ABB RobotStudio station: Solution15.rsstn

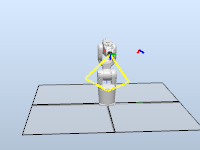
Station Solution15 (saved by RobotStudio 21.4.9700.0)
Controller IRB1200_7_70_1_LONG
  mechanical unit ROB_1: IRB1200_7_70_STD_03, 6 joints, base frame (0, 0, 0) mm
Layout (positions relative to the parent item):
  - IRB1200_7_70_STD_03 [mechanism, from Robots\IRB1200_7_70_STD_03.rslib] at (0, 0, 0) mm; joint values [-0.0012, -0.0017, 0.0867, -0.015, -0.085, 0.0148] (rad or m)
Targets, tools, work objects and paths stored in the station, written as RAPID:
! task T_ROB1
MODULE Module1
  CONST robtarget Target_10:=[[422.014082513,0,750.099998965],[0.499999994,0,0.866025407,0],[0,0,0,0],[9E+09,9E+09,9E+09,9E+09,9E+09,9E+09]];
  CONST robtarget Target_20:=[[116.600967602,405.58611933,750.099998965],[0.399420887,-0.520949955,0.691817281,0.300770592],[0,0,-1,0],[9E+09,9E+09,9E+09,9E+09,9E+09,9E+09]];
  CONST jointtarget JointTarget_0:=[[-0.62,0.28,5.37,-6.22,-5.68,6.19],[9E+09,9E+09,9E+09,9E+09,9E+09,9E+09]];
  CONST jointtarget JointTarget_1:=[[-1.23,0.35,5.9,-11.16,-6.37,11.09],[9E+09,9E+09,9E+09,9E+09,9E+09,9E+09]];
  CONST jointtarget JointTarget_2:=[[-1.84,0.44,6.41,-15.11,-7.09,15],[9E+09,9E+09,9E+09,9E+09,9E+09,9E+09]];
  CONST jointtarget JointTarget_3:=[[-2.46,0.53,6.92,-18.33,-7.84,18.17],[9E+09,9E+09,9E+09,9E+09,9E+09,9E+09]];
  CONST jointtarget JointTarget_4:=[[-3.07,0.64,7.41,-20.97,-8.61,20.76],[9E+09,9E+09,9E+09,9E+09,9E+09,9E+09]];
  CONST jointtarget JointTarget_5:=[[-3.69,0.77,7.89,-23.18,-9.4,22.9],[9E+09,9E+09,9E+09,9E+09,9E+09,9E+09]];
  CONST jointtarget JointTarget_6:=[[-4.3,0.9,8.35,-25.05,-10.2,24.7],[9E+09,9E+09,9E+09,9E+09,9E+09,9E+09]];
  CONST jointtarget JointTarget_7:=[[-4.91,1.05,8.8,-26.64,-11,26.22],[9E+09,9E+09,9E+09,9E+09,9E+09,9E+09]];
  CONST jointtarget JointTarget_8:=[[-5.52,1.21,9.25,-28.02,-11.81,27.52],[9E+09,9E+09,9E+09,9E+09,9E+09,9E+09]];
  CONST jointtarget JointTarget_9:=[[-6.13,1.39,9.67,-29.23,-12.63,28.63],[9E+09,9E+09,9E+09,9E+09,9E+09,9E+09]];
  CONST jointtarget JointTarget_11:=[[-7.34,1.78,10.5,-31.22,-14.27,30.43],[9E+09,9E+09,9E+09,9E+09,9E+09,9E+09]];
  CONST jointtarget JointTarget_12:=[[-7.95,1.99,10.89,-32.06,-15.09,31.16],[9E+09,9E+09,9E+09,9E+09,9E+09,9E+09]];
  CONST jointtarget JointTarget_13:=[[-8.55,2.21,11.27,-32.81,-15.92,31.8],[9E+09,9E+09,9E+09,9E+09,9E+09,9E+09]];
  CONST jointtarget JointTarget_14:=[[-9.15,2.45,11.63,-33.5,-16.74,32.36],[9E+09,9E+09,9E+09,9E+09,9E+09,9E+09]];
  CONST jointtarget JointTarget_15:=[[-9.75,2.7,11.99,-34.12,-17.57,32.86],[9E+09,9E+09,9E+09,9E+09,9E+09,9E+09]];
  CONST jointtarget JointTarget_16:=[[-10.34,2.97,12.33,-34.68,-18.39,33.29],[9E+09,9E+09,9E+09,9E+09,9E+09,9E+09]];
  CONST jointtarget JointTarget_17:=[[-10.94,3.24,12.66,-35.2,-19.22,33.67],[9E+09,9E+09,9E+09,9E+09,9E+09,9E+09]];
  CONST jointtarget JointTarget_18:=[[-11.53,3.53,12.97,-35.69,-20.04,34.01],[9E+09,9E+09,9E+09,9E+09,9E+09,9E+09]];
  CONST jointtarget JointTarget_19:=[[-12.12,3.83,13.27,-36.13,-20.86,34.3],[9E+09,9E+09,9E+09,9E+09,9E+09,9E+09]];
  CONST jointtarget JointTarget_21:=[[-13.29,4.47,13.84,-36.94,-22.49,34.79],[9E+09,9E+09,9E+09,9E+09,9E+09,9E+09]];
  CONST jointtarget JointTarget_22:=[[-13.87,4.8,14.11,-37.31,-23.3,34.99],[9E+09,9E+09,9E+09,9E+09,9E+09,9E+09]];
  CONST jointtarget JointTarget_23:=[[-14.45,5.15,14.36,-37.65,-24.11,35.16],[9E+09,9E+09,9E+09,9E+09,9E+09,9E+09]];
  CONST jointtarget JointTarget_24:=[[-15.02,5.51,14.6,-37.98,-24.91,35.3],[9E+09,9E+09,9E+09,9E+09,9E+09,9E+09]];
  CONST jointtarget JointTarget_25:=[[-15.6,5.88,14.82,-38.29,-25.72,35.43],[9E+09,9E+09,9E+09,9E+09,9E+09,9E+09]];
  CONST jointtarget JointTarget_26:=[[-16.17,6.27,15.04,-38.59,-26.51,35.53],[9E+09,9E+09,9E+09,9E+09,9E+09,9E+09]];
  CONST jointtarget JointTarget_27:=[[-16.73,6.66,15.23,-38.87,-27.3,35.61],[9E+09,9E+09,9E+09,9E+09,9E+09,9E+09]];
  CONST jointtarget JointTarget_28:=[[-17.29,7.07,15.42,-39.15,-28.09,35.68],[9E+09,9E+09,9E+09,9E+09,9E+09,9E+09]];
  CONST jointtarget JointTarget_29:=[[-17.85,7.48,15.6,-39.41,-28.88,35.74],[9E+09,9E+09,9E+09,9E+09,9E+09,9E+09]];
  CONST jointtarget JointTarget_30:=[[-18.41,7.91,15.76,-39.67,-29.65,35.78],[9E+09,9E+09,9E+09,9E+09,9E+09,9E+09]];
  CONST jointtarget JointTarget_31:=[[-18.96,8.35,15.9,-39.91,-30.43,35.8],[9E+09,9E+09,9E+09,9E+09,9E+09,9E+09]];
  CONST jointtarget JointTarget_32:=[[-19.51,8.8,16.04,-40.15,-31.19,35.82],[9E+09,9E+09,9E+09,9E+09,9E+09,9E+09]];
  CONST jointtarget JointTarget_33:=[[-20.05,9.26,16.16,-40.39,-31.95,35.82],[9E+09,9E+09,9E+09,9E+09,9E+09,9E+09]];
  CONST jointtarget JointTarget_34:=[[-20.6,9.72,16.27,-40.61,-32.71,35.81],[9E+09,9E+09,9E+09,9E+09,9E+09,9E+09]];
  CONST jointtarget JointTarget_35:=[[-21.13,10.2,16.36,-40.84,-33.46,35.8],[9E+09,9E+09,9E+09,9E+09,9E+09,9E+09]];
  CONST jointtarget JointTarget_36:=[[-21.67,10.69,16.44,-41.06,-34.2,35.77],[9E+09,9E+09,9E+09,9E+09,9E+09,9E+09]];
  CONST jointtarget JointTarget_37:=[[-22.19,11.19,16.51,-41.28,-34.93,35.74],[9E+09,9E+09,9E+09,9E+09,9E+09,9E+09]];
  CONST jointtarget JointTarget_38:=[[-22.72,11.7,16.56,-41.49,-35.66,35.7],[9E+09,9E+09,9E+09,9E+09,9E+09,9E+09]];
  CONST jointtarget JointTarget_39:=[[-23.24,12.21,16.6,-41.7,-36.38,35.65],[9E+09,9E+09,9E+09,9E+09,9E+09,9E+09]];
  CONST jointtarget JointTarget_40:=[[-23.76,12.74,16.63,-41.91,-37.1,35.6],[9E+09,9E+09,9E+09,9E+09,9E+09,9E+09]];
  CONST jointtarget JointTarget_41:=[[-24.27,13.27,16.65,-42.12,-37.8,35.54],[9E+09,9E+09,9E+09,9E+09,9E+09,9E+09]];
  CONST jointtarget JointTarget_42:=[[-24.78,13.81,16.65,-42.32,-38.5,35.48],[9E+09,9E+09,9E+09,9E+09,9E+09,9E+09]];
  CONST jointtarget JointTarget_43:=[[-25.29,14.36,16.64,-42.53,-39.19,35.41],[9E+09,9E+09,9E+09,9E+09,9E+09,9E+09]];
  CONST jointtarget JointTarget_44:=[[-25.79,14.92,16.61,-42.73,-39.87,35.34],[9E+09,9E+09,9E+09,9E+09,9E+09,9E+09]];
  CONST jointtarget JointTarget_45:=[[-26.28,15.49,16.57,-42.94,-40.55,35.26],[9E+09,9E+09,9E+09,9E+09,9E+09,9E+09]];
  CONST jointtarget JointTarget_46:=[[-26.78,16.06,16.52,-43.14,-41.21,35.18],[9E+09,9E+09,9E+09,9E+09,9E+09,9E+09]];
  CONST jointtarget JointTarget_47:=[[-27.26,16.64,16.45,-43.35,-41.87,35.1],[9E+09,9E+09,9E+09,9E+09,9E+09,9E+09]];
  CONST jointtarget JointTarget_48:=[[-27.75,17.23,16.37,-43.55,-42.51,35.02],[9E+09,9E+09,9E+09,9E+09,9E+09,9E+09]];
  CONST jointtarget JointTarget_49:=[[-28.23,17.82,16.28,-43.75,-43.15,34.93],[9E+09,9E+09,9E+09,9E+09,9E+09,9E+09]];
  CONST jointtarget JointTarget_50:=[[-28.7,18.42,16.18,-43.96,-43.78,34.84],[9E+09,9E+09,9E+09,9E+09,9E+09,9E+09]];
  CONST jointtarget JointTarget_51:=[[-29.17,19.03,16.06,-44.16,-44.4,34.76],[9E+09,9E+09,9E+09,9E+09,9E+09,9E+09]];
  CONST jointtarget JointTarget_52:=[[-29.64,19.65,15.93,-44.37,-45.01,34.66],[9E+09,9E+09,9E+09,9E+09,9E+09,9E+09]];
  CONST jointtarget JointTarget_53:=[[-30.1,20.27,15.78,-44.57,-45.61,34.57],[9E+09,9E+09,9E+09,9E+09,9E+09,9E+09]];
  CONST jointtarget JointTarget_54:=[[-30.56,20.89,15.62,-44.78,-46.21,34.48],[9E+09,9E+09,9E+09,9E+09,9E+09,9E+09]];
  CONST jointtarget JointTarget_55:=[[-31.02,21.52,15.45,-44.99,-46.79,34.39],[9E+09,9E+09,9E+09,9E+09,9E+09,9E+09]];
  CONST jointtarget JointTarget_56:=[[-31.47,22.16,15.27,-45.2,-47.36,34.3],[9E+09,9E+09,9E+09,9E+09,9E+09,9E+09]];
  CONST jointtarget JointTarget_57:=[[-31.91,22.8,15.07,-45.41,-47.92,34.21],[9E+09,9E+09,9E+09,9E+09,9E+09,9E+09]];
  CONST jointtarget JointTarget_58:=[[-32.35,23.44,14.86,-45.62,-48.48,34.12],[9E+09,9E+09,9E+09,9E+09,9E+09,9E+09]];
  CONST jointtarget JointTarget_59:=[[-32.79,24.09,14.63,-45.84,-49.02,34.03],[9E+09,9E+09,9E+09,9E+09,9E+09,9E+09]];
  CONST jointtarget JointTarget_60:=[[-33.22,24.75,14.4,-46.05,-49.55,33.94],[9E+09,9E+09,9E+09,9E+09,9E+09,9E+09]];
  CONST jointtarget JointTarget_61:=[[-33.65,25.41,14.15,-46.27,-50.07,33.86],[9E+09,9E+09,9E+09,9E+09,9E+09,9E+09]];
  CONST jointtarget JointTarget_62:=[[-34.07,26.07,13.89,-46.48,-50.59,33.77],[9E+09,9E+09,9E+09,9E+09,9E+09,9E+09]];
  CONST jointtarget JointTarget_63:=[[-34.49,26.74,13.61,-46.7,-51.09,33.69],[9E+09,9E+09,9E+09,9E+09,9E+09,9E+09]];
  CONST jointtarget JointTarget_64:=[[-34.91,27.41,13.32,-46.92,-51.58,33.61],[9E+09,9E+09,9E+09,9E+09,9E+09,9E+09]];
  CONST jointtarget JointTarget_65:=[[-35.32,28.08,13.02,-47.15,-52.06,33.53],[9E+09,9E+09,9E+09,9E+09,9E+09,9E+09]];
  CONST jointtarget JointTarget_66:=[[-35.73,28.76,12.71,-47.37,-52.53,33.46],[9E+09,9E+09,9E+09,9E+09,9E+09,9E+09]];
  CONST jointtarget JointTarget_67:=[[-36.13,29.44,12.38,-47.59,-53,33.38],[9E+09,9E+09,9E+09,9E+09,9E+09,9E+09]];
  CONST jointtarget JointTarget_68:=[[-36.53,30.13,12.04,-47.82,-53.45,33.31],[9E+09,9E+09,9E+09,9E+09,9E+09,9E+09]];
  CONST jointtarget JointTarget_69:=[[-36.93,30.81,11.69,-48.05,-53.89,33.25],[9E+09,9E+09,9E+09,9E+09,9E+09,9E+09]];
  CONST jointtarget JointTarget_70:=[[-37.32,31.5,11.33,-48.27,-54.32,33.19],[9E+09,9E+09,9E+09,9E+09,9E+09,9E+09]];
  CONST jointtarget JointTarget_71:=[[-37.7,32.19,10.95,-48.5,-54.74,33.13],[9E+09,9E+09,9E+09,9E+09,9E+09,9E+09]];
  CONST jointtarget JointTarget_72:=[[-38.09,32.89,10.56,-48.73,-55.15,33.07],[9E+09,9E+09,9E+09,9E+09,9E+09,9E+09]];
  CONST jointtarget JointTarget_73:=[[-38.47,33.59,10.16,-48.97,-55.55,33.02],[9E+09,9E+09,9E+09,9E+09,9E+09,9E+09]];
  CONST jointtarget JointTarget_74:=[[-38.84,34.28,9.74,-49.2,-55.94,32.98],[9E+09,9E+09,9E+09,9E+09,9E+09,9E+09]];
  CONST jointtarget JointTarget_75:=[[-38.67,34.05,10.66,-48.69,-56.3,32.26],[9E+09,9E+09,9E+09,9E+09,9E+09,9E+09]];
  CONST jointtarget JointTarget_76:=[[-38.5,33.82,11.57,-48.17,-56.66,31.55],[9E+09,9E+09,9E+09,9E+09,9E+09,9E+09]];
  CONST jointtarget JointTarget_77:=[[-38.33,33.6,12.48,-47.66,-57.03,30.85],[9E+09,9E+09,9E+09,9E+09,9E+09,9E+09]];
  CONST jointtarget JointTarget_78:=[[-38.15,33.4,13.37,-47.16,-57.41,30.15],[9E+09,9E+09,9E+09,9E+09,9E+09,9E+09]];
  CONST jointtarget JointTarget_79:=[[-37.97,33.2,14.26,-46.65,-57.79,29.45],[9E+09,9E+09,9E+09,9E+09,9E+09,9E+09]];
  CONST jointtarget JointTarget_80:=[[-37.79,33.01,15.14,-46.15,-58.18,28.76],[9E+09,9E+09,9E+09,9E+09,9E+09,9E+09]];
  CONST jointtarget JointTarget_81:=[[-37.6,32.82,16.01,-45.65,-58.57,28.08],[9E+09,9E+09,9E+09,9E+09,9E+09,9E+09]];
  CONST jointtarget JointTarget_82:=[[-37.41,32.65,16.88,-45.15,-58.97,27.4],[9E+09,9E+09,9E+09,9E+09,9E+09,9E+09]];
  CONST jointtarget JointTarget_83:=[[-37.22,32.49,17.73,-44.66,-59.37,26.72],[9E+09,9E+09,9E+09,9E+09,9E+09,9E+09]];
  CONST jointtarget JointTarget_84:=[[-37.02,32.34,18.58,-44.17,-59.78,26.06],[9E+09,9E+09,9E+09,9E+09,9E+09,9E+09]];
  CONST jointtarget JointTarget_85:=[[-36.81,32.19,19.43,-43.68,-60.19,25.39],[9E+09,9E+09,9E+09,9E+09,9E+09,9E+09]];
  CONST jointtarget JointTarget_86:=[[-36.61,32.06,20.26,-43.19,-60.61,24.73],[9E+09,9E+09,9E+09,9E+09,9E+09,9E+09]];
  CONST jointtarget JointTarget_87:=[[-36.4,31.93,21.09,-42.7,-61.04,24.08],[9E+09,9E+09,9E+09,9E+09,9E+09,9E+09]];
  CONST jointtarget JointTarget_88:=[[-36.18,31.81,21.91,-42.22,-61.47,23.43],[9E+09,9E+09,9E+09,9E+09,9E+09,9E+09]];
  CONST jointtarget JointTarget_89:=[[-35.96,31.71,22.72,-41.73,-61.91,22.78],[9E+09,9E+09,9E+09,9E+09,9E+09,9E+09]];
  CONST jointtarget JointTarget_90:=[[-35.74,31.61,23.53,-41.25,-62.36,22.14],[9E+09,9E+09,9E+09,9E+09,9E+09,9E+09]];
  CONST jointtarget JointTarget_91:=[[-35.51,31.53,24.33,-40.76,-62.81,21.5],[9E+09,9E+09,9E+09,9E+09,9E+09,9E+09]];
  CONST jointtarget JointTarget_92:=[[-35.27,31.45,25.12,-40.28,-63.27,20.87],[9E+09,9E+09,9E+09,9E+09,9E+09,9E+09]];
  CONST jointtarget JointTarget_93:=[[-35.03,31.38,25.91,-39.8,-63.74,20.24],[9E+09,9E+09,9E+09,9E+09,9E+09,9E+09]];
  CONST jointtarget JointTarget_94:=[[-34.79,31.33,26.69,-39.32,-64.21,19.61],[9E+09,9E+09,9E+09,9E+09,9E+09,9E+09]];
  CONST jointtarget JointTarget_95:=[[-34.54,31.29,27.46,-38.84,-64.7,18.99],[9E+09,9E+09,9E+09,9E+09,9E+09,9E+09]];
  CONST jointtarget JointTarget_96:=[[-34.28,31.25,28.22,-38.36,-65.19,18.37],[9E+09,9E+09,9E+09,9E+09,9E+09,9E+09]];
  CONST jointtarget JointTarget_97:=[[-34.02,31.23,28.98,-37.88,-65.69,17.76],[9E+09,9E+09,9E+09,9E+09,9E+09,9E+09]];
  CONST jointtarget JointTarget_98:=[[-33.76,31.22,29.73,-37.4,-66.19,17.15],[9E+09,9E+09,9E+09,9E+09,9E+09,9E+09]];
  CONST jointtarget JointTarget_99:=[[-33.48,31.23,30.47,-36.92,-66.71,16.54],[9E+09,9E+09,9E+09,9E+09,9E+09,9E+09]];
  CONST jointtarget JointTarget_100:=[[-33.2,31.24,31.21,-36.43,-67.23,15.94],[9E+09,9E+09,9E+09,9E+09,9E+09,9E+09]];
  CONST jointtarget JointTarget_101:=[[-32.92,31.27,31.94,-35.95,-67.76,15.35],[9E+09,9E+09,9E+09,9E+09,9E+09,9E+09]];
  CONST jointtarget JointTarget_102:=[[-32.62,31.31,32.66,-35.47,-68.31,14.75],[9E+09,9E+09,9E+09,9E+09,9E+09,9E+09]];
  CONST jointtarget JointTarget_103:=[[-32.32,31.36,33.38,-34.98,-68.86,14.16],[9E+09,9E+09,9E+09,9E+09,9E+09,9E+09]];
  CONST jointtarget JointTarget_104:=[[-32.02,31.42,34.08,-34.49,-69.42,13.58],[9E+09,9E+09,9E+09,9E+09,9E+09,9E+09]];
  CONST jointtarget JointTarget_105:=[[-31.7,31.5,34.78,-34.01,-69.99,13],[9E+09,9E+09,9E+09,9E+09,9E+09,9E+09]];
  CONST jointtarget JointTarget_106:=[[-31.38,31.59,35.48,-33.51,-70.57,12.42],[9E+09,9E+09,9E+09,9E+09,9E+09,9E+09]];
  CONST jointtarget JointTarget_107:=[[-31.05,31.7,36.16,-33.02,-71.16,11.85],[9E+09,9E+09,9E+09,9E+09,9E+09,9E+09]];
  CONST jointtarget JointTarget_108:=[[-30.71,31.82,36.84,-32.53,-71.77,11.28],[9E+09,9E+09,9E+09,9E+09,9E+09,9E+09]];
  CONST jointtarget JointTarget_109:=[[-30.36,31.95,37.51,-32.03,-72.38,10.72],[9E+09,9E+09,9E+09,9E+09,9E+09,9E+09]];
  CONST jointtarget JointTarget_110:=[[-30.01,32.1,38.17,-31.53,-73.01,10.17],[9E+09,9E+09,9E+09,9E+09,9E+09,9E+09]];
  CONST jointtarget JointTarget_111:=[[-29.64,32.27,38.83,-31.03,-73.64,9.61],[9E+09,9E+09,9E+09,9E+09,9E+09,9E+09]];
  CONST jointtarget JointTarget_112:=[[-29.27,32.45,39.47,-30.52,-74.29,9.07],[9E+09,9E+09,9E+09,9E+09,9E+09,9E+09]];
  CONST jointtarget JointTarget_113:=[[-28.88,32.65,40.11,-30.01,-74.96,8.53],[9E+09,9E+09,9E+09,9E+09,9E+09,9E+09]];
  CONST jointtarget JointTarget_114:=[[-28.49,32.86,40.74,-29.5,-75.63,7.99],[9E+09,9E+09,9E+09,9E+09,9E+09,9E+09]];
  CONST jointtarget JointTarget_115:=[[-28.08,33.09,41.36,-28.98,-76.32,7.46],[9E+09,9E+09,9E+09,9E+09,9E+09,9E+09]];
  CONST jointtarget JointTarget_116:=[[-27.67,33.33,41.97,-28.46,-77.02,6.94],[9E+09,9E+09,9E+09,9E+09,9E+09,9E+09]];
  CONST jointtarget JointTarget_117:=[[-27.24,33.6,42.57,-27.93,-77.73,6.43],[9E+09,9E+09,9E+09,9E+09,9E+09,9E+09]];
  CONST jointtarget JointTarget_118:=[[-26.8,33.88,43.17,-27.4,-78.46,5.92],[9E+09,9E+09,9E+09,9E+09,9E+09,9E+09]];
  CONST jointtarget JointTarget_119:=[[-26.35,34.18,43.75,-26.86,-79.2,5.42],[9E+09,9E+09,9E+09,9E+09,9E+09,9E+09]];
  CONST jointtarget JointTarget_120:=[[-25.89,34.49,44.33,-26.32,-79.96,4.93],[9E+09,9E+09,9E+09,9E+09,9E+09,9E+09]];
  CONST jointtarget JointTarget_121:=[[-25.41,34.83,44.89,-25.77,-80.73,4.45],[9E+09,9E+09,9E+09,9E+09,9E+09,9E+09]];
  CONST jointtarget JointTarget_122:=[[-24.92,35.18,45.45,-25.21,-81.51,3.98],[9E+09,9E+09,9E+09,9E+09,9E+09,9E+09]];
  CONST jointtarget JointTarget_123:=[[-24.41,35.56,45.99,-24.65,-82.31,3.51],[9E+09,9E+09,9E+09,9E+09,9E+09,9E+09]];
  CONST jointtarget JointTarget_124:=[[-23.89,35.95,46.53,-24.08,-83.13,3.06],[9E+09,9E+09,9E+09,9E+09,9E+09,9E+09]];
  CONST jointtarget JointTarget_125:=[[-23.36,36.36,47.05,-23.5,-83.96,2.62],[9E+09,9E+09,9E+09,9E+09,9E+09,9E+09]];
  CONST jointtarget JointTarget_126:=[[-22.81,36.79,47.56,-22.91,-84.8,2.19],[9E+09,9E+09,9E+09,9E+09,9E+09,9E+09]];
  CONST jointtarget JointTarget_127:=[[-22.24,37.25,48.06,-22.31,-85.66,1.78],[9E+09,9E+09,9E+09,9E+09,9E+09,9E+09]];
  CONST jointtarget JointTarget_128:=[[-21.66,37.72,48.55,-21.7,-86.54,1.38],[9E+09,9E+09,9E+09,9E+09,9E+09,9E+09]];
  CONST jointtarget JointTarget_129:=[[-21.05,38.21,49.03,-21.08,-87.43,0.99],[9E+09,9E+09,9E+09,9E+09,9E+09,9E+09]];
  CONST jointtarget JointTarget_130:=[[-20.43,38.73,49.5,-20.44,-88.34,0.62],[9E+09,9E+09,9E+09,9E+09,9E+09,9E+09]];
  CONST jointtarget JointTarget_131:=[[-19.79,39.26,49.95,-19.8,-89.26,0.27],[9E+09,9E+09,9E+09,9E+09,9E+09,9E+09]];
  CONST jointtarget JointTarget_132:=[[-19.13,39.81,50.39,-19.13,-90.19,-0.07],[9E+09,9E+09,9E+09,9E+09,9E+09,9E+09]];
  CONST jointtarget JointTarget_133:=[[-18.45,40.39,50.82,-18.46,-91.15,-0.38],[9E+09,9E+09,9E+09,9E+09,9E+09,9E+09]];
  CONST jointtarget JointTarget_134:=[[-17.75,40.98,51.23,-17.76,-92.11,-0.68],[9E+09,9E+09,9E+09,9E+09,9E+09,9E+09]];
  CONST jointtarget JointTarget_135:=[[-17.03,41.6,51.63,-17.05,-93.09,-0.95],[9E+09,9E+09,9E+09,9E+09,9E+09,9E+09]];
  CONST jointtarget JointTarget_136:=[[-16.28,42.24,52.02,-16.32,-94.08,-1.19],[9E+09,9E+09,9E+09,9E+09,9E+09,9E+09]];
  CONST jointtarget JointTarget_137:=[[-15.51,42.89,52.39,-15.57,-95.08,-1.41],[9E+09,9E+09,9E+09,9E+09,9E+09,9E+09]];
  CONST jointtarget JointTarget_138:=[[-14.72,43.56,52.74,-14.8,-96.1,-1.61],[9E+09,9E+09,9E+09,9E+09,9E+09,9E+09]];
  CONST jointtarget JointTarget_139:=[[-13.89,44.26,53.08,-14,-97.12,-1.77],[9E+09,9E+09,9E+09,9E+09,9E+09,9E+09]];
  CONST jointtarget JointTarget_140:=[[-13.05,44.97,53.41,-13.18,-98.16,-1.9],[9E+09,9E+09,9E+09,9E+09,9E+09,9E+09]];
  CONST jointtarget JointTarget_141:=[[-12.17,45.7,53.72,-12.33,-99.2,-2],[9E+09,9E+09,9E+09,9E+09,9E+09,9E+09]];
  CONST jointtarget JointTarget_142:=[[-11.27,46.44,54.01,-11.45,-100.25,-2.06],[9E+09,9E+09,9E+09,9E+09,9E+09,9E+09]];
  CONST jointtarget JointTarget_143:=[[-10.33,47.2,54.28,-10.54,-101.3,-2.09],[9E+09,9E+09,9E+09,9E+09,9E+09,9E+09]];
  CONST jointtarget JointTarget_144:=[[-9.37,47.98,54.54,-9.6,-102.35,-2.07],[9E+09,9E+09,9E+09,9E+09,9E+09,9E+09]];
  CONST jointtarget JointTarget_145:=[[-8.38,48.76,54.78,-8.61,-103.4,-2.01],[9E+09,9E+09,9E+09,9E+09,9E+09,9E+09]];
  CONST jointtarget JointTarget_146:=[[-7.35,49.57,55.01,-7.59,-104.45,-1.91],[9E+09,9E+09,9E+09,9E+09,9E+09,9E+09]];
  CONST jointtarget JointTarget_147:=[[-6.29,50.38,55.21,-6.53,-105.5,-1.75],[9E+09,9E+09,9E+09,9E+09,9E+09,9E+09]];
  CONST jointtarget JointTarget_148:=[[-5.2,51.2,55.4,-5.42,-106.53,-1.55],[9E+09,9E+09,9E+09,9E+09,9E+09,9E+09]];
  CONST jointtarget JointTarget_149:=[[-4.07,52.03,55.57,-4.27,-107.56,-1.29],[9E+09,9E+09,9E+09,9E+09,9E+09,9E+09]];
  CONST jointtarget JointTarget_150:=[[-3.04,51.52,55.51,-3.17,-107.01,-0.93],[9E+09,9E+09,9E+09,9E+09,9E+09,9E+09]];
  CONST jointtarget JointTarget_151:=[[-2.02,51.02,55.45,-2.1,-106.45,-0.6],[9E+09,9E+09,9E+09,9E+09,9E+09,9E+09]];
  CONST jointtarget JointTarget_152:=[[-1.02,50.51,55.37,-1.06,-105.87,-0.29],[9E+09,9E+09,9E+09,9E+09,9E+09,9E+09]];
  CONST jointtarget JointTarget_153:=[[-0.03,50,55.28,-0.03,-105.28,-0.01],[9E+09,9E+09,9E+09,9E+09,9E+09,9E+09]];
  CONST jointtarget JointTarget_154:=[[0.93,49.49,55.18,0.97,-104.67,0.24],[9E+09,9E+09,9E+09,9E+09,9E+09,9E+09]];
  CONST jointtarget JointTarget_155:=[[1.88,48.99,55.07,1.94,-104.04,0.47],[9E+09,9E+09,9E+09,9E+09,9E+09,9E+09]];
  CONST jointtarget JointTarget_156:=[[2.82,48.48,54.94,2.9,-103.41,0.67],[9E+09,9E+09,9E+09,9E+09,9E+09,9E+09]];
  CONST jointtarget JointTarget_157:=[[3.73,47.98,54.81,3.83,-102.76,0.85],[9E+09,9E+09,9E+09,9E+09,9E+09,9E+09]];
  CONST jointtarget JointTarget_158:=[[4.63,47.48,54.67,4.73,-102.11,1],[9E+09,9E+09,9E+09,9E+09,9E+09,9E+09]];
  CONST jointtarget JointTarget_159:=[[5.51,46.99,54.52,5.62,-101.45,1.12],[9E+09,9E+09,9E+09,9E+09,9E+09,9E+09]];
  CONST jointtarget JointTarget_160:=[[6.37,46.5,54.35,6.49,-100.78,1.22],[9E+09,9E+09,9E+09,9E+09,9E+09,9E+09]];
  CONST jointtarget JointTarget_161:=[[7.22,46.01,54.18,7.33,-100.11,1.29],[9E+09,9E+09,9E+09,9E+09,9E+09,9E+09]];
  CONST jointtarget JointTarget_162:=[[8.05,45.53,54,8.16,-99.43,1.35],[9E+09,9E+09,9E+09,9E+09,9E+09,9E+09]];
  CONST jointtarget JointTarget_163:=[[8.86,45.06,53.8,8.97,-98.75,1.38],[9E+09,9E+09,9E+09,9E+09,9E+09,9E+09]];
  CONST jointtarget JointTarget_164:=[[9.66,44.59,53.6,9.76,-98.07,1.38],[9E+09,9E+09,9E+09,9E+09,9E+09,9E+09]];
  CONST jointtarget JointTarget_165:=[[10.44,44.13,53.39,10.53,-97.39,1.37],[9E+09,9E+09,9E+09,9E+09,9E+09,9E+09]];
  CONST jointtarget JointTarget_166:=[[11.2,43.68,53.17,11.28,-96.71,1.34],[9E+09,9E+09,9E+09,9E+09,9E+09,9E+09]];
  CONST jointtarget JointTarget_167:=[[11.95,43.23,52.93,12.02,-96.03,1.28],[9E+09,9E+09,9E+09,9E+09,9E+09,9E+09]];
  CONST jointtarget JointTarget_168:=[[12.68,42.79,52.69,12.74,-95.35,1.21],[9E+09,9E+09,9E+09,9E+09,9E+09,9E+09]];
  CONST jointtarget JointTarget_169:=[[13.4,42.36,52.45,13.44,-94.67,1.12],[9E+09,9E+09,9E+09,9E+09,9E+09,9E+09]];
  CONST jointtarget JointTarget_170:=[[14.1,41.94,52.19,14.14,-94,1.01],[9E+09,9E+09,9E+09,9E+09,9E+09,9E+09]];
  CONST jointtarget JointTarget_171:=[[14.79,41.52,51.92,14.81,-93.33,0.88],[9E+09,9E+09,9E+09,9E+09,9E+09,9E+09]];
  CONST jointtarget JointTarget_172:=[[15.46,41.12,51.65,15.48,-92.66,0.74],[9E+09,9E+09,9E+09,9E+09,9E+09,9E+09]];
  CONST jointtarget JointTarget_173:=[[16.12,40.72,51.36,16.13,-92,0.58],[9E+09,9E+09,9E+09,9E+09,9E+09,9E+09]];
  CONST jointtarget JointTarget_174:=[[16.76,40.34,51.07,16.77,-91.35,0.41],[9E+09,9E+09,9E+09,9E+09,9E+09,9E+09]];
  CONST jointtarget JointTarget_175:=[[17.39,39.96,50.77,17.39,-90.7,0.22],[9E+09,9E+09,9E+09,9E+09,9E+09,9E+09]];
  CONST jointtarget JointTarget_176:=[[18.01,39.59,50.46,18.01,-90.05,0.02],[9E+09,9E+09,9E+09,9E+09,9E+09,9E+09]];
  CONST jointtarget JointTarget_177:=[[18.61,39.23,50.15,18.61,-89.41,-0.2],[9E+09,9E+09,9E+09,9E+09,9E+09,9E+09]];
  CONST jointtarget JointTarget_178:=[[19.2,38.89,49.82,19.21,-88.78,-0.42],[9E+09,9E+09,9E+09,9E+09,9E+09,9E+09]];
  CONST jointtarget JointTarget_179:=[[19.78,38.55,49.49,19.79,-88.15,-0.66],[9E+09,9E+09,9E+09,9E+09,9E+09,9E+09]];
  CONST jointtarget JointTarget_180:=[[20.35,38.22,49.15,20.37,-87.54,-0.91],[9E+09,9E+09,9E+09,9E+09,9E+09,9E+09]];
  CONST jointtarget JointTarget_181:=[[20.9,37.9,48.81,20.93,-86.93,-1.18],[9E+09,9E+09,9E+09,9E+09,9E+09,9E+09]];
  CONST jointtarget JointTarget_182:=[[21.44,37.59,48.46,21.49,-86.32,-1.45],[9E+09,9E+09,9E+09,9E+09,9E+09,9E+09]];
  CONST jointtarget JointTarget_183:=[[21.97,37.29,48.1,22.04,-85.72,-1.73],[9E+09,9E+09,9E+09,9E+09,9E+09,9E+09]];
  CONST jointtarget JointTarget_184:=[[22.49,37,47.73,22.58,-85.14,-2.02],[9E+09,9E+09,9E+09,9E+09,9E+09,9E+09]];
  CONST jointtarget JointTarget_185:=[[23,36.72,47.36,23.11,-84.55,-2.32],[9E+09,9E+09,9E+09,9E+09,9E+09,9E+09]];
  CONST jointtarget JointTarget_186:=[[23.5,36.46,46.98,23.64,-83.98,-2.63],[9E+09,9E+09,9E+09,9E+09,9E+09,9E+09]];
  CONST jointtarget JointTarget_187:=[[23.99,36.2,46.59,24.16,-83.41,-2.94],[9E+09,9E+09,9E+09,9E+09,9E+09,9E+09]];
  CONST jointtarget JointTarget_188:=[[24.46,35.95,46.2,24.67,-82.86,-3.27],[9E+09,9E+09,9E+09,9E+09,9E+09,9E+09]];
  CONST jointtarget JointTarget_189:=[[24.93,35.71,45.8,25.17,-82.3,-3.6],[9E+09,9E+09,9E+09,9E+09,9E+09,9E+09]];
  CONST jointtarget JointTarget_190:=[[25.39,35.48,45.4,25.67,-81.76,-3.94],[9E+09,9E+09,9E+09,9E+09,9E+09,9E+09]];
  CONST jointtarget JointTarget_191:=[[25.84,35.26,44.98,26.17,-81.23,-4.29],[9E+09,9E+09,9E+09,9E+09,9E+09,9E+09]];
  CONST jointtarget JointTarget_192:=[[26.28,35.05,44.57,26.65,-80.7,-4.64],[9E+09,9E+09,9E+09,9E+09,9E+09,9E+09]];
  CONST jointtarget JointTarget_193:=[[26.71,34.85,44.15,27.14,-80.18,-5],[9E+09,9E+09,9E+09,9E+09,9E+09,9E+09]];
  CONST jointtarget JointTarget_194:=[[27.13,34.65,43.72,27.61,-79.67,-5.36],[9E+09,9E+09,9E+09,9E+09,9E+09,9E+09]];
  CONST jointtarget JointTarget_195:=[[27.54,34.47,43.28,28.09,-79.16,-5.73],[9E+09,9E+09,9E+09,9E+09,9E+09,9E+09]];
  CONST jointtarget JointTarget_196:=[[27.95,34.3,42.84,28.55,-78.66,-6.11],[9E+09,9E+09,9E+09,9E+09,9E+09,9E+09]];
  CONST jointtarget JointTarget_197:=[[28.34,34.13,42.4,29.02,-78.17,-6.49],[9E+09,9E+09,9E+09,9E+09,9E+09,9E+09]];
  CONST jointtarget JointTarget_198:=[[28.73,33.98,41.95,29.47,-77.69,-6.87],[9E+09,9E+09,9E+09,9E+09,9E+09,9E+09]];
  CONST jointtarget JointTarget_199:=[[29.11,33.83,41.5,29.93,-77.22,-7.26],[9E+09,9E+09,9E+09,9E+09,9E+09,9E+09]];
  CONST jointtarget JointTarget_200:=[[29.49,33.69,41.03,30.38,-76.75,-7.65],[9E+09,9E+09,9E+09,9E+09,9E+09,9E+09]];
  CONST jointtarget JointTarget_201:=[[29.85,33.57,40.57,30.82,-76.28,-8.05],[9E+09,9E+09,9E+09,9E+09,9E+09,9E+09]];
  CONST jointtarget JointTarget_202:=[[30.21,33.44,40.1,31.26,-75.83,-8.45],[9E+09,9E+09,9E+09,9E+09,9E+09,9E+09]];
  CONST jointtarget JointTarget_203:=[[30.56,33.33,39.62,31.7,-75.38,-8.86],[9E+09,9E+09,9E+09,9E+09,9E+09,9E+09]];
  CONST jointtarget JointTarget_204:=[[30.91,33.23,39.14,32.14,-74.94,-9.27],[9E+09,9E+09,9E+09,9E+09,9E+09,9E+09]];
  CONST jointtarget JointTarget_205:=[[31.25,33.13,38.66,32.57,-74.51,-9.68],[9E+09,9E+09,9E+09,9E+09,9E+09,9E+09]];
  CONST jointtarget JointTarget_206:=[[31.58,33.04,38.17,33,-74.08,-10.1],[9E+09,9E+09,9E+09,9E+09,9E+09,9E+09]];
  CONST jointtarget JointTarget_207:=[[31.91,32.96,37.68,33.42,-73.66,-10.52],[9E+09,9E+09,9E+09,9E+09,9E+09,9E+09]];
  CONST jointtarget JointTarget_208:=[[32.23,32.89,37.18,33.84,-73.24,-10.94],[9E+09,9E+09,9E+09,9E+09,9E+09,9E+09]];
  CONST jointtarget JointTarget_209:=[[32.54,32.83,36.67,34.26,-72.83,-11.37],[9E+09,9E+09,9E+09,9E+09,9E+09,9E+09]];
  CONST jointtarget JointTarget_210:=[[32.85,32.77,36.17,34.68,-72.43,-11.8],[9E+09,9E+09,9E+09,9E+09,9E+09,9E+09]];
  CONST jointtarget JointTarget_211:=[[33.15,32.72,35.65,35.09,-72.03,-12.23],[9E+09,9E+09,9E+09,9E+09,9E+09,9E+09]];
  CONST jointtarget JointTarget_212:=[[33.45,32.68,35.14,35.5,-71.64,-12.67],[9E+09,9E+09,9E+09,9E+09,9E+09,9E+09]];
  CONST jointtarget JointTarget_213:=[[33.74,32.64,34.62,35.91,-71.25,-13.1],[9E+09,9E+09,9E+09,9E+09,9E+09,9E+09]];
  CONST jointtarget JointTarget_214:=[[34.03,32.62,34.09,36.32,-70.87,-13.54],[9E+09,9E+09,9E+09,9E+09,9E+09,9E+09]];
  CONST jointtarget JointTarget_215:=[[34.31,32.6,33.56,36.72,-70.49,-13.99],[9E+09,9E+09,9E+09,9E+09,9E+09,9E+09]];
  CONST jointtarget JointTarget_216:=[[34.58,32.58,33.03,37.12,-70.12,-14.43],[9E+09,9E+09,9E+09,9E+09,9E+09,9E+09]];
  CONST jointtarget JointTarget_217:=[[34.85,32.58,32.49,37.52,-69.76,-14.88],[9E+09,9E+09,9E+09,9E+09,9E+09,9E+09]];
  CONST jointtarget JointTarget_218:=[[35.12,32.58,31.95,37.92,-69.4,-15.33],[9E+09,9E+09,9E+09,9E+09,9E+09,9E+09]];
  CONST jointtarget JointTarget_219:=[[35.38,32.58,31.4,38.32,-69.04,-15.78],[9E+09,9E+09,9E+09,9E+09,9E+09,9E+09]];
  CONST jointtarget JointTarget_220:=[[35.64,32.59,30.85,38.71,-68.69,-16.24],[9E+09,9E+09,9E+09,9E+09,9E+09,9E+09]];
  CONST jointtarget JointTarget_221:=[[35.89,32.61,30.29,39.11,-68.35,-16.69],[9E+09,9E+09,9E+09,9E+09,9E+09,9E+09]];
  CONST jointtarget JointTarget_222:=[[36.14,32.64,29.73,39.5,-68.01,-17.15],[9E+09,9E+09,9E+09,9E+09,9E+09,9E+09]];
  CONST jointtarget JointTarget_223:=[[36.38,32.67,29.17,39.89,-67.67,-17.62],[9E+09,9E+09,9E+09,9E+09,9E+09,9E+09]];
  CONST jointtarget JointTarget_224:=[[36.62,32.71,28.6,40.28,-67.34,-18.08],[9E+09,9E+09,9E+09,9E+09,9E+09,9E+09]];
  CONST jointtarget JointTarget_225:=[[36.17,31.89,28.82,39.98,-66.74,-18.32],[9E+09,9E+09,9E+09,9E+09,9E+09,9E+09]];
  CONST jointtarget JointTarget_226:=[[35.73,31.08,29.02,39.68,-66.13,-18.56],[9E+09,9E+09,9E+09,9E+09,9E+09,9E+09]];
  CONST jointtarget JointTarget_227:=[[35.28,30.27,29.21,39.39,-65.51,-18.8],[9E+09,9E+09,9E+09,9E+09,9E+09,9E+09]];
  CONST jointtarget JointTarget_228:=[[34.82,29.46,29.39,39.1,-64.87,-19.04],[9E+09,9E+09,9E+09,9E+09,9E+09,9E+09]];
  CONST jointtarget JointTarget_229:=[[34.37,28.66,29.55,38.82,-64.22,-19.28],[9E+09,9E+09,9E+09,9E+09,9E+09,9E+09]];
  CONST jointtarget JointTarget_230:=[[33.91,27.86,29.69,38.54,-63.56,-19.53],[9E+09,9E+09,9E+09,9E+09,9E+09,9E+09]];
  CONST jointtarget JointTarget_231:=[[33.45,27.07,29.82,38.26,-62.89,-19.77],[9E+09,9E+09,9E+09,9E+09,9E+09,9E+09]];
  CONST jointtarget JointTarget_232:=[[32.99,26.28,29.94,37.99,-62.2,-20.01],[9E+09,9E+09,9E+09,9E+09,9E+09,9E+09]];
  CONST jointtarget JointTarget_233:=[[32.52,25.5,30.04,37.72,-61.5,-20.26],[9E+09,9E+09,9E+09,9E+09,9E+09,9E+09]];
  CONST jointtarget JointTarget_234:=[[32.05,24.72,30.12,37.45,-60.78,-20.5],[9E+09,9E+09,9E+09,9E+09,9E+09,9E+09]];
  CONST jointtarget JointTarget_235:=[[31.58,23.95,30.19,37.19,-60.06,-20.74],[9E+09,9E+09,9E+09,9E+09,9E+09,9E+09]];
  CONST jointtarget JointTarget_236:=[[31.11,23.18,30.24,36.93,-59.32,-20.98],[9E+09,9E+09,9E+09,9E+09,9E+09,9E+09]];
  CONST jointtarget JointTarget_237:=[[30.64,22.42,30.28,36.67,-58.58,-21.21],[9E+09,9E+09,9E+09,9E+09,9E+09,9E+09]];
  CONST jointtarget JointTarget_238:=[[30.16,21.67,30.3,36.42,-57.82,-21.45],[9E+09,9E+09,9E+09,9E+09,9E+09,9E+09]];
  CONST jointtarget JointTarget_239:=[[29.68,20.93,30.31,36.17,-57.05,-21.68],[9E+09,9E+09,9E+09,9E+09,9E+09,9E+09]];
  CONST jointtarget JointTarget_240:=[[29.2,20.2,30.3,35.92,-56.27,-21.91],[9E+09,9E+09,9E+09,9E+09,9E+09,9E+09]];
  CONST jointtarget JointTarget_241:=[[28.72,19.47,30.28,35.68,-55.49,-22.14],[9E+09,9E+09,9E+09,9E+09,9E+09,9E+09]];
  CONST jointtarget JointTarget_242:=[[28.24,18.76,30.24,35.44,-54.69,-22.36],[9E+09,9E+09,9E+09,9E+09,9E+09,9E+09]];
  CONST jointtarget JointTarget_243:=[[27.75,18.05,30.18,35.2,-53.88,-22.58],[9E+09,9E+09,9E+09,9E+09,9E+09,9E+09]];
  CONST jointtarget JointTarget_244:=[[27.27,17.35,30.11,34.97,-53.07,-22.79],[9E+09,9E+09,9E+09,9E+09,9E+09,9E+09]];
  CONST jointtarget JointTarget_245:=[[26.78,16.67,30.03,34.74,-52.24,-23.01],[9E+09,9E+09,9E+09,9E+09,9E+09,9E+09]];
  CONST jointtarget JointTarget_246:=[[26.29,15.99,29.93,34.51,-51.41,-23.21],[9E+09,9E+09,9E+09,9E+09,9E+09,9E+09]];
  CONST jointtarget JointTarget_247:=[[25.79,15.33,29.81,34.29,-50.57,-23.41],[9E+09,9E+09,9E+09,9E+09,9E+09,9E+09]];
  CONST jointtarget JointTarget_248:=[[25.3,14.67,29.68,34.07,-49.73,-23.61],[9E+09,9E+09,9E+09,9E+09,9E+09,9E+09]];
  CONST jointtarget JointTarget_249:=[[24.81,14.03,29.54,33.85,-48.88,-23.8],[9E+09,9E+09,9E+09,9E+09,9E+09,9E+09]];
  CONST jointtarget JointTarget_250:=[[24.31,13.4,29.38,33.63,-48.02,-23.99],[9E+09,9E+09,9E+09,9E+09,9E+09,9E+09]];
  CONST jointtarget JointTarget_251:=[[23.81,12.78,29.2,33.42,-47.15,-24.16],[9E+09,9E+09,9E+09,9E+09,9E+09,9E+09]];
  CONST jointtarget JointTarget_252:=[[23.31,12.18,29.01,33.2,-46.28,-24.34],[9E+09,9E+09,9E+09,9E+09,9E+09,9E+09]];
  CONST jointtarget JointTarget_253:=[[22.81,11.58,28.8,32.99,-45.41,-24.5],[9E+09,9E+09,9E+09,9E+09,9E+09,9E+09]];
  CONST jointtarget JointTarget_254:=[[22.31,11,28.58,32.78,-44.53,-24.66],[9E+09,9E+09,9E+09,9E+09,9E+09,9E+09]];
  CONST jointtarget JointTarget_255:=[[21.81,10.44,28.35,32.57,-43.64,-24.81],[9E+09,9E+09,9E+09,9E+09,9E+09,9E+09]];
  CONST jointtarget JointTarget_256:=[[21.31,9.88,28.1,32.37,-42.75,-24.96],[9E+09,9E+09,9E+09,9E+09,9E+09,9E+09]];
  CONST jointtarget JointTarget_257:=[[20.81,9.35,27.84,32.16,-41.86,-25.09],[9E+09,9E+09,9E+09,9E+09,9E+09,9E+09]];
  CONST jointtarget JointTarget_258:=[[20.3,8.82,27.56,31.95,-40.97,-25.22],[9E+09,9E+09,9E+09,9E+09,9E+09,9E+09]];
  CONST jointtarget JointTarget_259:=[[19.8,8.31,27.27,31.75,-40.07,-25.34],[9E+09,9E+09,9E+09,9E+09,9E+09,9E+09]];
  CONST jointtarget JointTarget_260:=[[19.29,7.81,26.96,31.54,-39.17,-25.45],[9E+09,9E+09,9E+09,9E+09,9E+09,9E+09]];
  CONST jointtarget JointTarget_261:=[[18.78,7.33,26.64,31.33,-38.26,-25.55],[9E+09,9E+09,9E+09,9E+09,9E+09,9E+09]];
  CONST jointtarget JointTarget_262:=[[18.28,6.86,26.3,31.12,-37.36,-25.64],[9E+09,9E+09,9E+09,9E+09,9E+09,9E+09]];
  CONST jointtarget JointTarget_263:=[[17.77,6.41,25.96,30.91,-36.45,-25.72],[9E+09,9E+09,9E+09,9E+09,9E+09,9E+09]];
  CONST jointtarget JointTarget_264:=[[17.26,5.97,25.59,30.7,-35.54,-25.79],[9E+09,9E+09,9E+09,9E+09,9E+09,9E+09]];
  CONST jointtarget JointTarget_265:=[[16.76,5.55,25.22,30.48,-34.63,-25.84],[9E+09,9E+09,9E+09,9E+09,9E+09,9E+09]];
  CONST jointtarget JointTarget_266:=[[16.25,5.14,24.83,30.26,-33.72,-25.89],[9E+09,9E+09,9E+09,9E+09,9E+09,9E+09]];
  CONST jointtarget JointTarget_267:=[[15.74,4.74,24.43,30.04,-32.81,-25.92],[9E+09,9E+09,9E+09,9E+09,9E+09,9E+09]];
  CONST jointtarget JointTarget_268:=[[15.23,4.36,24.01,29.81,-31.9,-25.94],[9E+09,9E+09,9E+09,9E+09,9E+09,9E+09]];
  CONST jointtarget JointTarget_269:=[[14.73,4,23.58,29.58,-30.99,-25.95],[9E+09,9E+09,9E+09,9E+09,9E+09,9E+09]];
  CONST jointtarget JointTarget_270:=[[14.22,3.65,23.14,29.34,-30.08,-25.94],[9E+09,9E+09,9E+09,9E+09,9E+09,9E+09]];
  CONST jointtarget JointTarget_271:=[[13.71,3.32,22.68,29.1,-29.17,-25.92],[9E+09,9E+09,9E+09,9E+09,9E+09,9E+09]];
  CONST jointtarget JointTarget_272:=[[13.21,3,22.22,28.85,-28.26,-25.88],[9E+09,9E+09,9E+09,9E+09,9E+09,9E+09]];
  CONST jointtarget JointTarget_273:=[[12.7,2.7,21.73,28.58,-27.35,-25.82],[9E+09,9E+09,9E+09,9E+09,9E+09,9E+09]];
  CONST jointtarget JointTarget_274:=[[12.19,2.41,21.24,28.31,-26.45,-25.75],[9E+09,9E+09,9E+09,9E+09,9E+09,9E+09]];
  CONST jointtarget JointTarget_275:=[[11.69,2.13,20.74,28.03,-25.54,-25.65],[9E+09,9E+09,9E+09,9E+09,9E+09,9E+09]];
  CONST jointtarget JointTarget_276:=[[11.18,1.88,20.22,27.73,-24.63,-25.54],[9E+09,9E+09,9E+09,9E+09,9E+09,9E+09]];
  CONST jointtarget JointTarget_277:=[[10.68,1.63,19.69,27.42,-23.73,-25.4],[9E+09,9E+09,9E+09,9E+09,9E+09,9E+09]];
  CONST jointtarget JointTarget_278:=[[10.18,1.4,19.14,27.09,-22.83,-25.24],[9E+09,9E+09,9E+09,9E+09,9E+09,9E+09]];
  CONST jointtarget JointTarget_279:=[[9.67,1.19,18.59,26.74,-21.93,-25.05],[9E+09,9E+09,9E+09,9E+09,9E+09,9E+09]];
  CONST jointtarget JointTarget_280:=[[9.17,0.99,18.02,26.37,-21.03,-24.83],[9E+09,9E+09,9E+09,9E+09,9E+09,9E+09]];
  CONST jointtarget JointTarget_281:=[[8.67,0.81,17.44,25.98,-20.14,-24.58],[9E+09,9E+09,9E+09,9E+09,9E+09,9E+09]];
  CONST jointtarget JointTarget_282:=[[8.17,0.64,16.85,25.55,-19.25,-24.29],[9E+09,9E+09,9E+09,9E+09,9E+09,9E+09]];
  CONST jointtarget JointTarget_283:=[[7.68,0.48,16.25,25.1,-18.36,-23.97],[9E+09,9E+09,9E+09,9E+09,9E+09,9E+09]];
  CONST jointtarget JointTarget_284:=[[7.18,0.34,15.63,24.6,-17.47,-23.59],[9E+09,9E+09,9E+09,9E+09,9E+09,9E+09]];
  CONST jointtarget JointTarget_285:=[[6.69,0.21,15,24.06,-16.59,-23.17],[9E+09,9E+09,9E+09,9E+09,9E+09,9E+09]];
  CONST jointtarget JointTarget_286:=[[6.19,0.1,14.36,23.48,-15.71,-22.69],[9E+09,9E+09,9E+09,9E+09,9E+09,9E+09]];
  CONST jointtarget JointTarget_287:=[[5.7,0,13.71,22.83,-14.83,-22.14],[9E+09,9E+09,9E+09,9E+09,9E+09,9E+09]];
  CONST jointtarget JointTarget_288:=[[5.21,-0.08,13.05,22.11,-13.96,-21.51],[9E+09,9E+09,9E+09,9E+09,9E+09,9E+09]];
  CONST jointtarget JointTarget_289:=[[4.72,-0.15,12.37,21.3,-13.09,-20.79],[9E+09,9E+09,9E+09,9E+09,9E+09,9E+09]];
  CONST jointtarget JointTarget_290:=[[4.23,-0.21,11.69,20.39,-12.23,-19.97],[9E+09,9E+09,9E+09,9E+09,9E+09,9E+09]];
  CONST jointtarget JointTarget_291:=[[3.75,-0.25,10.99,19.36,-11.37,-19],[9E+09,9E+09,9E+09,9E+09,9E+09,9E+09]];
  CONST jointtarget JointTarget_292:=[[3.26,-0.28,10.28,18.17,-10.51,-17.88],[9E+09,9E+09,9E+09,9E+09,9E+09,9E+09]];
  CONST jointtarget JointTarget_293:=[[2.78,-0.29,9.55,16.78,-9.67,-16.56],[9E+09,9E+09,9E+09,9E+09,9E+09,9E+09]];
  CONST jointtarget JointTarget_294:=[[2.3,-0.29,8.82,15.15,-8.83,-14.98],[9E+09,9E+09,9E+09,9E+09,9E+09,9E+09]];
  CONST jointtarget JointTarget_295:=[[1.82,-0.28,8.07,13.19,-8,-13.07],[9E+09,9E+09,9E+09,9E+09,9E+09,9E+09]];
  CONST jointtarget JointTarget_296:=[[1.34,-0.25,7.32,10.81,-7.19,-10.72],[9E+09,9E+09,9E+09,9E+09,9E+09,9E+09]];
  CONST jointtarget JointTarget_297:=[[0.87,-0.22,6.55,7.84,-6.39,-7.79],[9E+09,9E+09,9E+09,9E+09,9E+09,9E+09]];
  CONST jointtarget JointTarget_298:=[[0.4,-0.16,5.76,4.07,-5.61,-4.05],[9E+09,9E+09,9E+09,9E+09,9E+09,9E+09]];
  CONST jointtarget JointTarget_299:=[[-0.07,-0.1,4.97,-0.86,-4.87,0.85],[9E+09,9E+09,9E+09,9E+09,9E+09,9E+09]];
  CONST jointtarget JointTarget_10:=[[-6.74,1.58,10.09,-30.28,-13.45,29.6],[9E+09,9E+09,9E+09,9E+09,9E+09,9E+09]];
  CONST jointtarget JointTarget_20:=[[-12.71,4.14,13.56,-36.55,-21.67,34.56],[9E+09,9E+09,9E+09,9E+09,9E+09,9E+09]];
  PROC Path_10()
    MoveAbsJ JointTarget_0,v100,z1,tool0\WObj:=wobj0;
    MoveAbsJ JointTarget_1,v100,z1,tool0\WObj:=wobj0;
    MoveAbsJ JointTarget_2,v100,z1,tool0\WObj:=wobj0;
    MoveAbsJ JointTarget_3,v100,z1,tool0\WObj:=wobj0;
    MoveAbsJ JointTarget_4,v100,z1,tool0\WObj:=wobj0;
    MoveAbsJ JointTarget_5,v100,z1,tool0\WObj:=wobj0;
    MoveAbsJ JointTarget_6,v100,z1,tool0\WObj:=wobj0;
    MoveAbsJ JointTarget_7,v100,z1,tool0\WObj:=wobj0;
    MoveAbsJ JointTarget_8,v100,z1,tool0\WObj:=wobj0;
    MoveAbsJ JointTarget_9,v100,z1,tool0\WObj:=wobj0;
    MoveAbsJ JointTarget_10,v100,z1,tool0\WObj:=wobj0;
    MoveAbsJ JointTarget_11,v100,z1,tool0\WObj:=wobj0;
    MoveAbsJ JointTarget_12,v100,z1,tool0\WObj:=wobj0;
    MoveAbsJ JointTarget_13,v100,z1,tool0\WObj:=wobj0;
    MoveAbsJ JointTarget_14,v100,z1,tool0\WObj:=wobj0;
    MoveAbsJ JointTarget_15,v100,z1,tool0\WObj:=wobj0;
    MoveAbsJ JointTarget_16,v100,z1,tool0\WObj:=wobj0;
    MoveAbsJ JointTarget_17,v100,z1,tool0\WObj:=wobj0;
    MoveAbsJ JointTarget_18,v100,z1,tool0\WObj:=wobj0;
    MoveAbsJ JointTarget_19,v100,z1,tool0\WObj:=wobj0;
    MoveAbsJ JointTarget_20,v100,z1,tool0\WObj:=wobj0;
    MoveAbsJ JointTarget_21,v100,z1,tool0\WObj:=wobj0;
    MoveAbsJ JointTarget_22,v100,z1,tool0\WObj:=wobj0;
    MoveAbsJ JointTarget_23,v100,z1,tool0\WObj:=wobj0;
    MoveAbsJ JointTarget_24,v100,z1,tool0\WObj:=wobj0;
    MoveAbsJ JointTarget_25,v100,z1,tool0\WObj:=wobj0;
    MoveAbsJ JointTarget_26,v100,z1,tool0\WObj:=wobj0;
    MoveAbsJ JointTarget_27,v100,z1,tool0\WObj:=wobj0;
    MoveAbsJ JointTarget_28,v100,z1,tool0\WObj:=wobj0;
    MoveAbsJ JointTarget_29,v100,z1,tool0\WObj:=wobj0;
    MoveAbsJ JointTarget_30,v100,z1,tool0\WObj:=wobj0;
    MoveAbsJ JointTarget_31,v100,z1,tool0\WObj:=wobj0;
    MoveAbsJ JointTarget_32,v100,z1,tool0\WObj:=wobj0;
    MoveAbsJ JointTarget_33,v100,z1,tool0\WObj:=wobj0;
    MoveAbsJ JointTarget_34,v100,z1,tool0\WObj:=wobj0;
    MoveAbsJ JointTarget_35,v100,z1,tool0\WObj:=wobj0;
    MoveAbsJ JointTarget_36,v100,z1,tool0\WObj:=wobj0;
    MoveAbsJ JointTarget_37,v100,z1,tool0\WObj:=wobj0;
    MoveAbsJ JointTarget_38,v100,z1,tool0\WObj:=wobj0;
    MoveAbsJ JointTarget_39,v100,z1,tool0\WObj:=wobj0;
    MoveAbsJ JointTarget_40,v100,z1,tool0\WObj:=wobj0;
    MoveAbsJ JointTarget_41,v100,z1,tool0\WObj:=wobj0;
    MoveAbsJ JointTarget_42,v100,z1,tool0\WObj:=wobj0;
    MoveAbsJ JointTarget_43,v100,z1,tool0\WObj:=wobj0;
    MoveAbsJ JointTarget_44,v100,z1,tool0\WObj:=wobj0;
    MoveAbsJ JointTarget_45,v100,z1,tool0\WObj:=wobj0;
    MoveAbsJ JointTarget_46,v100,z1,tool0\WObj:=wobj0;
    MoveAbsJ JointTarget_47,v100,z1,tool0\WObj:=wobj0;
    MoveAbsJ JointTarget_48,v100,z1,tool0\WObj:=wobj0;
    MoveAbsJ JointTarget_49,v100,z1,tool0\WObj:=wobj0;
    MoveAbsJ JointTarget_50,v100,z1,tool0\WObj:=wobj0;
    MoveAbsJ JointTarget_51,v100,z1,tool0\WObj:=wobj0;
    MoveAbsJ JointTarget_52,v100,z1,tool0\WObj:=wobj0;
    MoveAbsJ JointTarget_53,v100,z1,tool0\WObj:=wobj0;
    MoveAbsJ JointTarget_54,v100,z1,tool0\WObj:=wobj0;
    MoveAbsJ JointTarget_55,v100,z1,tool0\WObj:=wobj0;
    MoveAbsJ JointTarget_56,v100,z1,tool0\WObj:=wobj0;
    MoveAbsJ JointTarget_57,v100,z1,tool0\WObj:=wobj0;
    MoveAbsJ JointTarget_58,v100,z1,tool0\WObj:=wobj0;
    MoveAbsJ JointTarget_59,v100,z1,tool0\WObj:=wobj0;
    MoveAbsJ JointTarget_60,v100,z1,tool0\WObj:=wobj0;
    MoveAbsJ JointTarget_61,v100,z1,tool0\WObj:=wobj0;
    MoveAbsJ JointTarget_62,v100,z1,tool0\WObj:=wobj0;
    MoveAbsJ JointTarget_63,v100,z1,tool0\WObj:=wobj0;
    MoveAbsJ JointTarget_64,v100,z1,tool0\WObj:=wobj0;
    MoveAbsJ JointTarget_65,v100,z1,tool0\WObj:=wobj0;
    MoveAbsJ JointTarget_66,v100,z1,tool0\WObj:=wobj0;
    MoveAbsJ JointTarget_67,v100,z1,tool0\WObj:=wobj0;
    MoveAbsJ JointTarget_68,v100,z1,tool0\WObj:=wobj0;
    MoveAbsJ JointTarget_69,v100,z1,tool0\WObj:=wobj0;
    MoveAbsJ JointTarget_70,v100,z1,tool0\WObj:=wobj0;
    MoveAbsJ JointTarget_71,v100,z1,tool0\WObj:=wobj0;
    MoveAbsJ JointTarget_72,v100,z1,tool0\WObj:=wobj0;
    MoveAbsJ JointTarget_73,v100,z1,tool0\WObj:=wobj0;
    MoveAbsJ JointTarget_74,v100,z1,tool0\WObj:=wobj0;
    MoveAbsJ JointTarget_75,v100,z1,tool0\WObj:=wobj0;
    MoveAbsJ JointTarget_76,v100,z1,tool0\WObj:=wobj0;
    MoveAbsJ JointTarget_77,v100,z1,tool0\WObj:=wobj0;
    MoveAbsJ JointTarget_78,v100,z1,tool0\WObj:=wobj0;
    MoveAbsJ JointTarget_79,v100,z1,tool0\WObj:=wobj0;
    MoveAbsJ JointTarget_80,v100,z1,tool0\WObj:=wobj0;
    MoveAbsJ JointTarget_81,v100,z1,tool0\WObj:=wobj0;
    MoveAbsJ JointTarget_82,v100,z1,tool0\WObj:=wobj0;
    MoveAbsJ JointTarget_83,v100,z1,tool0\WObj:=wobj0;
    MoveAbsJ JointTarget_84,v100,z1,tool0\WObj:=wobj0;
    MoveAbsJ JointTarget_85,v100,z1,tool0\WObj:=wobj0;
    MoveAbsJ JointTarget_86,v100,z1,tool0\WObj:=wobj0;
    MoveAbsJ JointTarget_87,v100,z1,tool0\WObj:=wobj0;
    MoveAbsJ JointTarget_88,v100,z1,tool0\WObj:=wobj0;
    MoveAbsJ JointTarget_89,v100,z1,tool0\WObj:=wobj0;
    MoveAbsJ JointTarget_90,v100,z1,tool0\WObj:=wobj0;
    MoveAbsJ JointTarget_91,v100,z1,tool0\WObj:=wobj0;
    MoveAbsJ JointTarget_92,v100,z1,tool0\WObj:=wobj0;
    MoveAbsJ JointTarget_93,v100,z1,tool0\WObj:=wobj0;
    MoveAbsJ JointTarget_94,v100,z1,tool0\WObj:=wobj0;
    MoveAbsJ JointTarget_95,v100,z1,tool0\WObj:=wobj0;
    MoveAbsJ JointTarget_96,v100,z1,tool0\WObj:=wobj0;
    MoveAbsJ JointTarget_97,v100,z1,tool0\WObj:=wobj0;
    MoveAbsJ JointTarget_98,v100,z1,tool0\WObj:=wobj0;
    MoveAbsJ JointTarget_99,v100,z1,tool0\WObj:=wobj0;
    MoveAbsJ JointTarget_100,v100,z1,tool0\WObj:=wobj0;
    MoveAbsJ JointTarget_101,v100,z1,tool0\WObj:=wobj0;
    MoveAbsJ JointTarget_102,v100,z1,tool0\WObj:=wobj0;
    MoveAbsJ JointTarget_103,v100,z1,tool0\WObj:=wobj0;
    MoveAbsJ JointTarget_104,v100,z1,tool0\WObj:=wobj0;
    MoveAbsJ JointTarget_105,v100,z1,tool0\WObj:=wobj0;
    MoveAbsJ JointTarget_106,v100,z1,tool0\WObj:=wobj0;
    MoveAbsJ JointTarget_107,v100,z1,tool0\WObj:=wobj0;
    MoveAbsJ JointTarget_108,v100,z1,tool0\WObj:=wobj0;
    MoveAbsJ JointTarget_109,v100,z1,tool0\WObj:=wobj0;
    MoveAbsJ JointTarget_110,v100,z1,tool0\WObj:=wobj0;
    MoveAbsJ JointTarget_111,v100,z1,tool0\WObj:=wobj0;
    MoveAbsJ JointTarget_112,v100,z1,tool0\WObj:=wobj0;
    MoveAbsJ JointTarget_113,v100,z1,tool0\WObj:=wobj0;
    MoveAbsJ JointTarget_114,v100,z1,tool0\WObj:=wobj0;
    MoveAbsJ JointTarget_115,v100,z1,tool0\WObj:=wobj0;
    MoveAbsJ JointTarget_116,v100,z1,tool0\WObj:=wobj0;
    MoveAbsJ JointTarget_117,v100,z1,tool0\WObj:=wobj0;
    MoveAbsJ JointTarget_118,v100,z1,tool0\WObj:=wobj0;
    MoveAbsJ JointTarget_119,v100,z1,tool0\WObj:=wobj0;
    MoveAbsJ JointTarget_120,v100,z1,tool0\WObj:=wobj0;
    MoveAbsJ JointTarget_121,v100,z1,tool0\WObj:=wobj0;
    MoveAbsJ JointTarget_122,v100,z1,tool0\WObj:=wobj0;
    MoveAbsJ JointTarget_123,v100,z1,tool0\WObj:=wobj0;
    MoveAbsJ JointTarget_124,v100,z1,tool0\WObj:=wobj0;
    MoveAbsJ JointTarget_125,v100,z1,tool0\WObj:=wobj0;
    MoveAbsJ JointTarget_126,v100,z1,tool0\WObj:=wobj0;
    MoveAbsJ JointTarget_127,v100,z1,tool0\WObj:=wobj0;
    MoveAbsJ JointTarget_128,v100,z1,tool0\WObj:=wobj0;
    MoveAbsJ JointTarget_129,v100,z1,tool0\WObj:=wobj0;
    MoveAbsJ JointTarget_130,v100,z1,tool0\WObj:=wobj0;
    MoveAbsJ JointTarget_131,v100,z1,tool0\WObj:=wobj0;
    MoveAbsJ JointTarget_132,v100,z1,tool0\WObj:=wobj0;
    MoveAbsJ JointTarget_133,v100,z1,tool0\WObj:=wobj0;
    MoveAbsJ JointTarget_134,v100,z1,tool0\WObj:=wobj0;
    MoveAbsJ JointTarget_135,v100,z1,tool0\WObj:=wobj0;
    MoveAbsJ JointTarget_136,v100,z1,tool0\WObj:=wobj0;
    MoveAbsJ JointTarget_137,v100,z1,tool0\WObj:=wobj0;
    MoveAbsJ JointTarget_138,v100,z1,tool0\WObj:=wobj0;
    MoveAbsJ JointTarget_139,v100,z1,tool0\WObj:=wobj0;
    MoveAbsJ JointTarget_140,v100,z1,tool0\WObj:=wobj0;
    MoveAbsJ JointTarget_141,v100,z1,tool0\WObj:=wobj0;
    MoveAbsJ JointTarget_142,v100,z1,tool0\WObj:=wobj0;
    MoveAbsJ JointTarget_143,v100,z1,tool0\WObj:=wobj0;
    MoveAbsJ JointTarget_144,v100,z1,tool0\WObj:=wobj0;
    MoveAbsJ JointTarget_145,v100,z1,tool0\WObj:=wobj0;
    MoveAbsJ JointTarget_146,v100,z1,tool0\WObj:=wobj0;
    MoveAbsJ JointTarget_147,v100,z1,tool0\WObj:=wobj0;
    MoveAbsJ JointTarget_148,v100,z1,tool0\WObj:=wobj0;
    MoveAbsJ JointTarget_149,v100,z1,tool0\WObj:=wobj0;
    MoveAbsJ JointTarget_150,v100,z1,tool0\WObj:=wobj0;
    MoveAbsJ JointTarget_151,v100,z1,tool0\WObj:=wobj0;
    MoveAbsJ JointTarget_152,v100,z1,tool0\WObj:=wobj0;
    MoveAbsJ JointTarget_153,v100,z1,tool0\WObj:=wobj0;
    MoveAbsJ JointTarget_154,v100,z1,tool0\WObj:=wobj0;
    MoveAbsJ JointTarget_155,v100,z1,tool0\WObj:=wobj0;
    MoveAbsJ JointTarget_156,v100,z1,tool0\WObj:=wobj0;
    MoveAbsJ JointTarget_157,v100,z1,tool0\WObj:=wobj0;
    MoveAbsJ JointTarget_158,v100,z1,tool0\WObj:=wobj0;
    MoveAbsJ JointTarget_159,v100,z1,tool0\WObj:=wobj0;
    MoveAbsJ JointTarget_160,v100,z1,tool0\WObj:=wobj0;
    MoveAbsJ JointTarget_161,v100,z1,tool0\WObj:=wobj0;
    MoveAbsJ JointTarget_162,v100,z1,tool0\WObj:=wobj0;
    MoveAbsJ JointTarget_163,v100,z1,tool0\WObj:=wobj0;
    MoveAbsJ JointTarget_164,v100,z1,tool0\WObj:=wobj0;
    MoveAbsJ JointTarget_165,v100,z1,tool0\WObj:=wobj0;
    MoveAbsJ JointTarget_166,v100,z1,tool0\WObj:=wobj0;
    MoveAbsJ JointTarget_167,v100,z1,tool0\WObj:=wobj0;
    MoveAbsJ JointTarget_168,v100,z1,tool0\WObj:=wobj0;
    MoveAbsJ JointTarget_169,v100,z1,tool0\WObj:=wobj0;
    MoveAbsJ JointTarget_170,v100,z1,tool0\WObj:=wobj0;
    MoveAbsJ JointTarget_171,v100,z1,tool0\WObj:=wobj0;
    MoveAbsJ JointTarget_172,v100,z1,tool0\WObj:=wobj0;
    MoveAbsJ JointTarget_173,v100,z1,tool0\WObj:=wobj0;
    MoveAbsJ JointTarget_174,v100,z1,tool0\WObj:=wobj0;
    MoveAbsJ JointTarget_175,v100,z1,tool0\WObj:=wobj0;
    MoveAbsJ JointTarget_176,v100,z1,tool0\WObj:=wobj0;
    MoveAbsJ JointTarget_177,v100,z1,tool0\WObj:=wobj0;
    MoveAbsJ JointTarget_178,v100,z1,tool0\WObj:=wobj0;
    MoveAbsJ JointTarget_179,v100,z1,tool0\WObj:=wobj0;
    MoveAbsJ JointTarget_180,v100,z1,tool0\WObj:=wobj0;
    MoveAbsJ JointTarget_181,v100,z1,tool0\WObj:=wobj0;
    MoveAbsJ JointTarget_182,v100,z1,tool0\WObj:=wobj0;
    MoveAbsJ JointTarget_183,v100,z1,tool0\WObj:=wobj0;
    MoveAbsJ JointTarget_184,v100,z1,tool0\WObj:=wobj0;
    MoveAbsJ JointTarget_185,v100,z1,tool0\WObj:=wobj0;
    MoveAbsJ JointTarget_186,v100,z1,tool0\WObj:=wobj0;
    MoveAbsJ JointTarget_187,v100,z1,tool0\WObj:=wobj0;
    MoveAbsJ JointTarget_188,v100,z1,tool0\WObj:=wobj0;
    MoveAbsJ JointTarget_189,v100,z1,tool0\WObj:=wobj0;
    MoveAbsJ JointTarget_190,v100,z1,tool0\WObj:=wobj0;
    MoveAbsJ JointTarget_191,v100,z1,tool0\WObj:=wobj0;
    MoveAbsJ JointTarget_192,v100,z1,tool0\WObj:=wobj0;
    MoveAbsJ JointTarget_193,v100,z1,tool0\WObj:=wobj0;
    MoveAbsJ JointTarget_194,v100,z1,tool0\WObj:=wobj0;
    MoveAbsJ JointTarget_195,v100,z1,tool0\WObj:=wobj0;
    MoveAbsJ JointTarget_196,v100,z1,tool0\WObj:=wobj0;
    MoveAbsJ JointTarget_197,v100,z1,tool0\WObj:=wobj0;
    MoveAbsJ JointTarget_198,v100,z1,tool0\WObj:=wobj0;
    MoveAbsJ JointTarget_199,v100,z1,tool0\WObj:=wobj0;
    MoveAbsJ JointTarget_200,v100,z1,tool0\WObj:=wobj0;
    MoveAbsJ JointTarget_201,v100,z1,tool0\WObj:=wobj0;
    MoveAbsJ JointTarget_202,v100,z1,tool0\WObj:=wobj0;
    MoveAbsJ JointTarget_203,v100,z1,tool0\WObj:=wobj0;
    MoveAbsJ JointTarget_204,v100,z1,tool0\WObj:=wobj0;
    MoveAbsJ JointTarget_205,v100,z1,tool0\WObj:=wobj0;
    MoveAbsJ JointTarget_206,v100,z1,tool0\WObj:=wobj0;
    MoveAbsJ JointTarget_207,v100,z1,tool0\WObj:=wobj0;
    MoveAbsJ JointTarget_208,v100,z1,tool0\WObj:=wobj0;
    MoveAbsJ JointTarget_209,v100,z1,tool0\WObj:=wobj0;
    MoveAbsJ JointTarget_210,v100,z1,tool0\WObj:=wobj0;
    MoveAbsJ JointTarget_211,v100,z1,tool0\WObj:=wobj0;
    MoveAbsJ JointTarget_212,v100,z1,tool0\WObj:=wobj0;
    MoveAbsJ JointTarget_213,v100,z1,tool0\WObj:=wobj0;
    MoveAbsJ JointTarget_214,v100,z1,tool0\WObj:=wobj0;
    MoveAbsJ JointTarget_215,v100,z1,tool0\WObj:=wobj0;
    MoveAbsJ JointTarget_216,v100,z1,tool0\WObj:=wobj0;
    MoveAbsJ JointTarget_217,v100,z1,tool0\WObj:=wobj0;
    MoveAbsJ JointTarget_218,v100,z1,tool0\WObj:=wobj0;
    MoveAbsJ JointTarget_219,v100,z1,tool0\WObj:=wobj0;
    MoveAbsJ JointTarget_220,v100,z1,tool0\WObj:=wobj0;
    MoveAbsJ JointTarget_221,v100,z1,tool0\WObj:=wobj0;
    MoveAbsJ JointTarget_222,v100,z1,tool0\WObj:=wobj0;
    MoveAbsJ JointTarget_223,v100,z1,tool0\WObj:=wobj0;
    MoveAbsJ JointTarget_224,v100,z1,tool0\WObj:=wobj0;
    MoveAbsJ JointTarget_225,v100,z1,tool0\WObj:=wobj0;
    MoveAbsJ JointTarget_226,v100,z1,tool0\WObj:=wobj0;
    MoveAbsJ JointTarget_227,v100,z1,tool0\WObj:=wobj0;
    MoveAbsJ JointTarget_228,v100,z1,tool0\WObj:=wobj0;
    MoveAbsJ JointTarget_229,v100,z1,tool0\WObj:=wobj0;
    MoveAbsJ JointTarget_230,v100,z1,tool0\WObj:=wobj0;
    MoveAbsJ JointTarget_231,v100,z1,tool0\WObj:=wobj0;
    MoveAbsJ JointTarget_232,v100,z1,tool0\WObj:=wobj0;
    MoveAbsJ JointTarget_233,v100,z1,tool0\WObj:=wobj0;
    MoveAbsJ JointTarget_234,v100,z1,tool0\WObj:=wobj0;
    MoveAbsJ JointTarget_235,v100,z1,tool0\WObj:=wobj0;
    MoveAbsJ JointTarget_236,v100,z1,tool0\WObj:=wobj0;
    MoveAbsJ JointTarget_237,v100,z1,tool0\WObj:=wobj0;
    MoveAbsJ JointTarget_238,v100,z1,tool0\WObj:=wobj0;
    MoveAbsJ JointTarget_239,v100,z1,tool0\WObj:=wobj0;
    MoveAbsJ JointTarget_240,v100,z1,tool0\WObj:=wobj0;
    MoveAbsJ JointTarget_241,v100,z1,tool0\WObj:=wobj0;
    MoveAbsJ JointTarget_242,v100,z1,tool0\WObj:=wobj0;
    MoveAbsJ JointTarget_243,v100,z1,tool0\WObj:=wobj0;
    MoveAbsJ JointTarget_244,v100,z1,tool0\WObj:=wobj0;
    MoveAbsJ JointTarget_245,v100,z1,tool0\WObj:=wobj0;
    MoveAbsJ JointTarget_246,v100,z1,tool0\WObj:=wobj0;
    MoveAbsJ JointTarget_247,v100,z1,tool0\WObj:=wobj0;
    MoveAbsJ JointTarget_248,v100,z1,tool0\WObj:=wobj0;
    MoveAbsJ JointTarget_249,v100,z1,tool0\WObj:=wobj0;
    MoveAbsJ JointTarget_250,v100,z1,tool0\WObj:=wobj0;
    MoveAbsJ JointTarget_251,v100,z1,tool0\WObj:=wobj0;
    MoveAbsJ JointTarget_252,v100,z1,tool0\WObj:=wobj0;
    MoveAbsJ JointTarget_253,v100,z1,tool0\WObj:=wobj0;
    MoveAbsJ JointTarget_254,v100,z1,tool0\WObj:=wobj0;
    MoveAbsJ JointTarget_255,v100,z1,tool0\WObj:=wobj0;
    MoveAbsJ JointTarget_256,v100,z1,tool0\WObj:=wobj0;
    MoveAbsJ JointTarget_257,v100,z1,tool0\WObj:=wobj0;
    MoveAbsJ JointTarget_258,v100,z1,tool0\WObj:=wobj0;
    MoveAbsJ JointTarget_259,v100,z1,tool0\WObj:=wobj0;
    MoveAbsJ JointTarget_260,v100,z1,tool0\WObj:=wobj0;
    MoveAbsJ JointTarget_261,v100,z1,tool0\WObj:=wobj0;
    MoveAbsJ JointTarget_262,v100,z1,tool0\WObj:=wobj0;
    MoveAbsJ JointTarget_263,v100,z1,tool0\WObj:=wobj0;
    MoveAbsJ JointTarget_264,v100,z1,tool0\WObj:=wobj0;
    MoveAbsJ JointTarget_265,v100,z1,tool0\WObj:=wobj0;
    MoveAbsJ JointTarget_266,v100,z1,tool0\WObj:=wobj0;
    MoveAbsJ JointTarget_267,v100,z1,tool0\WObj:=wobj0;
    MoveAbsJ JointTarget_268,v100,z1,tool0\WObj:=wobj0;
    MoveAbsJ JointTarget_269,v100,z1,tool0\WObj:=wobj0;
    MoveAbsJ JointTarget_270,v100,z1,tool0\WObj:=wobj0;
    MoveAbsJ JointTarget_271,v100,z1,tool0\WObj:=wobj0;
    MoveAbsJ JointTarget_272,v100,z1,tool0\WObj:=wobj0;
    MoveAbsJ JointTarget_273,v100,z1,tool0\WObj:=wobj0;
    MoveAbsJ JointTarget_274,v100,z1,tool0\WObj:=wobj0;
    MoveAbsJ JointTarget_275,v100,z1,tool0\WObj:=wobj0;
    MoveAbsJ JointTarget_276,v100,z1,tool0\WObj:=wobj0;
    MoveAbsJ JointTarget_277,v100,z1,tool0\WObj:=wobj0;
    MoveAbsJ JointTarget_278,v100,z1,tool0\WObj:=wobj0;
    MoveAbsJ JointTarget_279,v100,z1,tool0\WObj:=wobj0;
    MoveAbsJ JointTarget_280,v100,z1,tool0\WObj:=wobj0;
    MoveAbsJ JointTarget_281,v100,z1,tool0\WObj:=wobj0;
    MoveAbsJ JointTarget_282,v100,z1,tool0\WObj:=wobj0;
    MoveAbsJ JointTarget_283,v100,z1,tool0\WObj:=wobj0;
    MoveAbsJ JointTarget_284,v100,z1,tool0\WObj:=wobj0;
    MoveAbsJ JointTarget_285,v100,z1,tool0\WObj:=wobj0;
    MoveAbsJ JointTarget_286,v100,z1,tool0\WObj:=wobj0;
    MoveAbsJ JointTarget_287,v100,z1,tool0\WObj:=wobj0;
    MoveAbsJ JointTarget_288,v100,z1,tool0\WObj:=wobj0;
    MoveAbsJ JointTarget_289,v100,z1,tool0\WObj:=wobj0;
    MoveAbsJ JointTarget_290,v100,z1,tool0\WObj:=wobj0;
    MoveAbsJ JointTarget_291,v100,z1,tool0\WObj:=wobj0;
    MoveAbsJ JointTarget_292,v100,z1,tool0\WObj:=wobj0;
    MoveAbsJ JointTarget_293,v100,z1,tool0\WObj:=wobj0;
    MoveAbsJ JointTarget_294,v100,z1,tool0\WObj:=wobj0;
    MoveAbsJ JointTarget_295,v100,z1,tool0\WObj:=wobj0;
    MoveAbsJ JointTarget_296,v100,z1,tool0\WObj:=wobj0;
    MoveAbsJ JointTarget_297,v100,z1,tool0\WObj:=wobj0;
    MoveAbsJ JointTarget_298,v100,z1,tool0\WObj:=wobj0;
    MoveAbsJ JointTarget_299,v100,z1,tool0\WObj:=wobj0;
  ENDPROC
  PROC main()
    Path_10;
  ENDPROC
ENDMODULE

